// TIA Portal V18 export
FUNCTION_BLOCK "MAN_DESCRETE_cycle"   // FB41, FBD
{ S7_Optimized_Access := 'TRUE' }
VERSION : 0.1
// stored: AutoNumber true, IsIECCheckEnabled false, IsRetainMemResEnabled false, MemoryReserve 100, SetENOAutomatically false, UDAEnableTagReadback false
   VAR_INPUT
      off_conditions : Bool;
      on_trigger : Bool;
   END_VAR
   VAR_OUTPUT
      motors_go_now_command : Bool;
   END_VAR
   VAR_IN_OUT
      sate : UInt;
   END_VAR
BEGIN

REGION Network 1
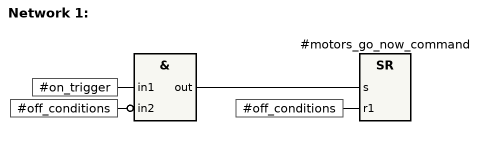
   IF #on_trigger AND NOT #off_conditions THEN
       #motors_go_now_command := TRUE;   // SR flip-flop
   END_IF;
   IF #off_conditions THEN #motors_go_now_command := FALSE; END_IF;
END_REGION
END_FUNCTION_BLOCK
